// TwinCAT 3 PLC project MonitoringSold
// ProgramVersion: 3.1.4024.0
// libraries:
//   Tc2_Standard, * (Beckhoff Automation GmbH)
//   Tc2_System, * (Beckhoff Automation GmbH)
//   Tc3_Module, * (Beckhoff Automation GmbH)
// project tree:
//   / PlcTask.TcTTO
//   POUs/ MAIN.TcPOU
//   _GENERAL/Functions/ FB_Predictive.TcPOU, FB_Statistic.TcPOU, STRUCT_StatisticsData.TcDUT
// real-time tasks:
//   TASK PlcTask: cycle T#10ms, priority 20, ADS port 350

CONFIGURATION MonitoringSold
    RESOURCE PLC ON TwinCAT3
        TASK PlcTask(INTERVAL := T#10ms, PRIORITY := 20);
        PROGRAM MAIN WITH PlcTask : MAIN;
    END_RESOURCE
END_CONFIGURATION

// ---- _GENERAL/Functions/STRUCT_StatisticsData.TcDUT
TYPE STRUCT_StatisticsData :
STRUCT
	udiCounter:UDINT:=1;
	udiCounterCoef:UDINT:=1;
	rStatCoefMin:REAL:=0.05;
	rStatCoef:REAL;
	rMinimum:REAL;
	rMaximum:REAL;
	rMean:REAL;
	rDevSum:REAL;
	rDev:REAL;
END_STRUCT
END_TYPE

// ---- POUs/MAIN.TcPOU
PROGRAM MAIN
VAR
END_VAR

END_PROGRAM

// ---- _GENERAL/Functions/FB_Predictive.TcPOU
FUNCTION_BLOCK FB_Predictive
VAR PERSISTENT
	rStatCoefMin:REAL:=0.0025;
	rFreqMean:REAL:=1.5;
	rFreqDev:REAL:=1.5;
END_VAR
VAR_INPUT
	bReset:BOOL;
END_VAR
VAR_OUTPUT
	bWarningMean:BOOL;
	bWarningDev:BOOL;
END_VAR
VAR
	fbStatistic:FB_Statistic;
	fbStatisticDev:FB_Statistic;
END_VAR

METHOD PRIVATE M_check
VAR_INPUT
END_VAR
IF THIS^.fbStatistic.bSaved THEN
	THIS^.bWarningMean	:= 	THIS^.fbStatistic.M_is_typical(freqTypical:=THIS^.rFreqMean);
	THIS^.bWarningDev 	:= 	THIS^.fbStatisticDev.M_is_typical(freqTypical:=THIS^.rFreqDev);
ELSE
	THIS^.bWarningMean:=FALSE;
	THIS^.bWarningDev:=FALSE;
END_IF
END_METHOD

METHOD M_run
VAR_INPUT
	rValue:REAL;
END_VAR
IF THIS^.bReset THEN
	THIS^.fbStatistic.bReset:=TRUE;
	THIS^.fbStatisticDev.bReset:=TRUE;
	THIS^.bReset:=FALSE;
END_IF

THIS^.fbStatistic.M_run(rStatCoefMin:=THIS^.rStatCoefMin,
						rCurrentValue:=rValue);
						
THIS^.fbStatisticDev.M_run(	rStatCoefMin:=THIS^.rStatCoefMin,
							rCurrentValue:=THIS^.fbStatistic.Data.rDev);
							
THIS^.M_check();
END_METHOD

END_FUNCTION_BLOCK

// ---- _GENERAL/Functions/FB_Statistic.TcPOU
FUNCTION_BLOCK FB_Statistic
VAR PERSISTENT
	bSaved:BOOL;
	Data:STRUCT_StatisticsData;
	DataSaved:STRUCT_StatisticsData;
	udiSamplesToSave:UDINT:=500;
	udiSamplesCounter:UDINT:=0;
END_VAR
VAR_INPUT
	bReset:BOOL;
	bRestore:BOOL;
END_VAR
VAR_OUTPUT
	rZScore:REAL;
END_VAR
VAR
	rValue:REAL;
END_VAR

METHOD PRIVATE M_calc_coef
VAR
	rCounter:REAL;
END_VAR
// Check counter and cast to real
IF THIS^.Data.udiCounter=0 THEN
	rCounter:=1;
END_IF
rCounter:=UDINT_TO_REAL(THIS^.Data.udiCounter);
// CALCULATE
// =======================================================
THIS^.Data.rStatCoef:=MAX((1/rCounter),THIS^.Data.rStatCoefMin);
// =======================================================
END_METHOD

METHOD PRIVATE M_calc_dev
VAR
	rRes:REAL;
END_VAR
IF THIS^.Data.rStatCoef=0 OR THIS^.Data.rStatCoef=1 THEN
	THIS^.Data.rDevSum:=0;
ELSE
	IF (THIS^.rValue-THIS^.Data.rMean)=0 THEN
		rRes:=0;
	ELSE
		rRes:=EXPT(THIS^.rValue-THIS^.Data.rMean,2);
	END_IF
	THIS^.Data.rDevSum :=	((1-THIS^.Data.rStatCoef)*THIS^.Data.rDevSum) + 
							(THIS^.Data.rStatCoef*rRes);
END_IF

IF THIS^.Data.rDevSum=0 THEN
	THIS^.Data.rDev:=0;
ELSE
	THIS^.Data.rDev:=SQRT(THIS^.Data.rDevSum);
END_IF
END_METHOD

METHOD PRIVATE M_calc_mean
VAR_INPUT
END_VAR
IF THIS^.Data.rStatCoef=1 THEN
	THIS^.Data.rMean:=THIS^.rValue;
ELSE
	IF THIS^.Data.rStatCoef<>0 THEN
		THIS^.Data.rMean := ((1-THIS^.Data.rStatCoef)*THIS^.Data.rMean) + 
							(THIS^.Data.rStatCoef*THIS^.rValue);
	end_if
END_IF
END_METHOD

METHOD PRIVATE M_calc_min_max
IF THIS^.Data.udiCounter=1 THEN
	THIS^.Data.rMaximum:=THIS^.rValue;
	THIS^.Data.rMinimum:=THIS^.rValue;
END_IF
THIS^.Data.rMinimum:=MIN(THIS^.Data.rMinimum,THIS^.rValue);
THIS^.Data.rMaximum:=MAX(THIS^.Data.rMaximum,THIS^.rValue);
END_METHOD

METHOD M_is_typical : BOOL	// >Return if the current value is in a typical frequence
VAR_INPUT
	freqTypical:REAL;		// Typical frequence
END_VAR
THIS^.rZScore := ABS((THIS^.Data.rMean - THIS^.DataSaved.rMean) / THIS^.DataSaved.rDev);
M_is_typical := THIS^.Data.rMean <= THIS^.DataSaved.rMean- (freqTypical*THIS^.DataSaved.rDev) OR
				THIS^.Data.rMean >= THIS^.DataSaved.rMean+ (freqTypical*THIS^.DataSaved.rDev);
END_METHOD

METHOD PRIVATE M_reset
IF THIS^.bReset THEN
	THIS^.Data.udiCounter:=1;
	THIS^.Data.rStatCoef:=0;
	THIS^.Data.rMinimum:=0;
	THIS^.Data.rMaximum:=0;
	THIS^.Data.rMean:=0;
	THIS^.Data.rDevSum:=0;
	THIS^.Data.rDev:=0;
	THIS^.bSaved:=FALSE;
	THIS^.udiSamplesCounter:=0;
	THIS^.bReset:=FALSE;
END_IF
END_METHOD

METHOD PRIVATE M_restore
VAR_INPUT
END_VAR
IF THIS^.bRestore THEN
	THIS^.Data := THIS^.DataSaved;
	THIS^.bRestore:=FALSE;
END_IF
END_METHOD

METHOD M_run
VAR_INPUT
	rStatCoefMin:REAL;
	rCurrentValue:REAL;
END_VAR
// Reset data
THIS^.M_reset();
// Restore data
THIS^.M_restore();
// Get current data
THIS^.Data.rStatCoefMin:=rStatCoefMin;
THIS^.rValue:=rCurrentValue;
// Calcs
THIS^.M_calc_coef();
THIS^.M_calc_min_max();
THIS^.M_calc_mean();
THIS^.M_calc_dev();
// Save data
THIS^.M_save();
// Update counter
IF THIS^.Data.udiCounter<4294967295 THEN
	THIS^.Data.udiCounter:=THIS^.Data.udiCounter+1;
END_IF
// Update coef counter until coef value if the minumum
IF THIS^.Data.rStatCoefMin<THIS^.Data.rStatCoef THEN
	THIS^.Data.udiCounterCoef:=THIS^.Data.udiCounterCoef+1;
END_IF
END_METHOD

METHOD PRIVATE M_save
IF NOT THIS^.bSaved THEN
	IF THIS^.udiSamplesCounter<THIS^.udiSamplesToSave THEN
		THIS^.udiSamplesCounter:=THIS^.udiSamplesCounter+1;
	ELSE
		THIS^.DataSaved:=THIS^.Data;
		THIS^.bSaved:=TRUE;
		THIS^.udiSamplesCounter:=0;
	END_IF
END_IF
END_METHOD

END_FUNCTION_BLOCK
